# EPICS alarm handler configuration: alh_files/mgnt_und.alhConfig
GROUP NULL MGNT:UND1:1
   $COMMAND edm -x -eolc -noedit mgnt_und1_main.edl

$ALIAS UND1
$GUIDANCE
und Magnet
   Group Name: MGNT:UND1:1
   Summary PV:  MGNT:UND1:1:STATSUMY
$END

   INCLUDE MGNT:UND1:1 ./mgnt_und1_bend.alhConfig
   INCLUDE MGNT:UND1:1 ./mgnt_und1_lgps.alhConfig
   INCLUDE MGNT:UND1:1 ./mgnt_und1_quad.alhConfig
   INCLUDE MGNT:UND1:1 ./mgnt_und1_xcor.alhConfig
   INCLUDE MGNT:UND1:1 ./mgnt_und1_ycor.alhConfig
